FUNCTION_BLOCK AOI_CylinderAdmin
VAR_INPUT
END_VAR
VAR_OUTPUT
	ActInTime: DINT;
	ActOutTime: DINT;
END_VAR
VAR
	TON_InCheck: TON;
	TON_OutCheck: TON;
	rtOUT: R_trig;
    rtIn: R_trig;
END_VAR
VAR_IN_OUT
	Admin: UDT_CylinderAdmin;
END_VAR

IF admin.i.mode=0 THEN
   IF admin.i.HmiIN THEN
	  admin.o.ValveIn:=TRUE;
	  admin.o.ValveOut:=FALSE;
   END_IF
   IF admin.i.HmiOUT THEN
	  admin.o.ValveIn:=FALSE;
	  admin.o.ValveOut:=TRUE;
   END_IF
END_IF
IF admin.i.mode=1 THEN
   IF admin.i.ActiveIn THEN
	  admin.o.ValveIn:=TRUE;
	  admin.o.ValveOut:=FALSE;
   END_IF
   IF admin.i.ActiveOut THEN
	  admin.o.ValveIn:=FALSE;
	  admin.o.ValveOut:=TRUE;
   END_IF
   IF NOT admin.i.ActiveIn AND NOT admin.i.ActiveOut  THEN
	  admin.o.ValveIn:=FALSE;
	  admin.o.ValveOut:=FALSE;
   END_IF
END_IF

TON_InCheck(IN:=admin.o.ValveIn AND NOT admin.i.Reset , PT:=DINT_TO_TIME(admin.i.CheckTime) , Q=> , ET=> );
TON_OutCheck(IN:=admin.o.ValveOut AND NOT admin.i.Reset, PT:=DINT_TO_TIME(admin.i.CheckTime) , Q=> , ET=> );
IF ton_incheck.Q AND NOT admin.i.InSensor THEN
   admin.o.Error:=TRUE;
END_IF
IF Ton_OutCheck.Q AND NOT admin.i.OutSensor THEN 
   admin.o.Error:=TRUE;
END_IF
IF admin.i.Reset THEN
   admin.o.Error:=FALSE;
END_IF

IF rtOUT.Q  AND NOT admin.o.Error THEN
   ActOutTime:=TIME_TO_DINT(TON_OutCheck.ET);
END_IF

IF rtIN.Q  AND NOT admin.o.Error THEN
   ActInTime:=TIME_TO_DINT(TON_InCheck.ET);
END_IF

rtOUT(CLK:= admin.i.OutSensor , Q=> );
rtIn(CLK:=  admin.i.InSensor, Q=> );

END_FUNCTION_BLOCK

(* stored: Version 1.1.0.1, ProductVersion 3.1.4022.16
   POU AOI_CylinderAdmin: Id {4163de3b-aae8-4b75-852a-b5be4cbd0661}, SpecialFunc None *)
